FUNCTION FC_BatCalculate : LREAL
VAR_INPUT
	lbatdata : LREAL;
END_VAR
VAR
END_VAR

FC_BatCalculate := ((3000-lbatdata)/3000)*100; // 1000 UDP

END_FUNCTION

(* stored: Version 1.1.0.1, ProductVersion 3.1.4024.13
   POU FC_BatCalculate: Id {efa77ea7-4b46-4dc8-9c66-7a0b2cd15977}, SpecialFunc None *)
